GLOBALCONSTANTS Funk_DI (* Funk_DI constants *)
  (* Standard: 61499-1; Description: Copyright (c) 2024 HR Agrartechnik GmbH This program and the accompanying materials are made available under the terms of the Eclipse Public License 2.0 which is available at https://www.eclipse.org/legal/epl-2.0/ SPDX-License-Identifier: EPL-2.0 *)
  (* Version 1.0, 2024-01-25, Franz Höpfinger, HR Agrartechnik GmbH *)
  PACKAGE Funk::io::DI;
  VAR_GLOBAL CONSTANT
    DigitalInput_Key_01 : Funk::io::DI::Funk_DI_S := (Pin := 1);
    DigitalInput_Key_02 : Funk::io::DI::Funk_DI_S := (Pin := 2);
    DigitalInput_Key_03 : Funk::io::DI::Funk_DI_S := (Pin := 3);
    DigitalInput_Key_04 : Funk::io::DI::Funk_DI_S := (Pin := 4);
    DigitalInput_Key_05 : Funk::io::DI::Funk_DI_S := (Pin := 5);
    DigitalInput_Key_06 : Funk::io::DI::Funk_DI_S := (Pin := 6);
    DigitalInput_Key_07 : Funk::io::DI::Funk_DI_S := (Pin := 7);
    DigitalInput_Key_08 : Funk::io::DI::Funk_DI_S := (Pin := 8);
    DigitalInput_Key_09 : Funk::io::DI::Funk_DI_S := (Pin := 9);
    DigitalInput_Key_10 : Funk::io::DI::Funk_DI_S := (Pin := 10);
    DigitalInput_Key_11 : Funk::io::DI::Funk_DI_S := (Pin := 11);
    DigitalInput_Key_12 : Funk::io::DI::Funk_DI_S := (Pin := 12);
    DigitalInput_Key_13 : Funk::io::DI::Funk_DI_S := (Pin := 13);
    DigitalInput_Key_14 : Funk::io::DI::Funk_DI_S := (Pin := 14);
    DigitalInput_Key_15 : Funk::io::DI::Funk_DI_S := (Pin := 15);
    DigitalInput_Key_START : Funk::io::DI::Funk_DI_S := (Pin := 25);
    DigitalInput_Key_STOP : Funk::io::DI::Funk_DI_S := (Pin := 0);
    DigitalInput_Key_STATUS : Funk::io::DI::Funk_DI_S := (Pin := -1);
    DigitalInput_Key_COUNTER : Funk::io::DI::Funk_DI_S := (Pin := -6);
    Invalid : Funk::io::DI::Funk_DI_S := (Pin := 127);
  END_VAR
END_GLOBALCONSTANTS
